INTERFACE I_DiagnosisEtherCATSlave

//エラー発生を出力
PROPERTY bError : BOOL
GET
END_GET
END_PROPERTY

//呼び出して診断実行
METHOD Execute
VAR_INPUT
END_VAR
END_METHOD

END_INTERFACE

(* stored: Version 1.1.0.1
   Itf I_DiagnosisEtherCATSlave: Id {090ab407-e917-4381-989f-025f06abcb34}
   Property bError: Id {cc5a4ad7-70c3-43c2-9131-4ee25fdc5989}
   Get Get: Id {12caa3ea-629a-4514-8762-74b9502c71f0}
   Method Execute: Id {e8bb91c4-88c5-42df-a91d-5249e670b9c9} *)
